ADAPTER IReactorData (* Adapter Interface *)
  (* Standard: 61499-1 *)
  (* Version 0.0, 7/4/2026, Schneider Electric *)
  PACKAGE SE.Nereda;
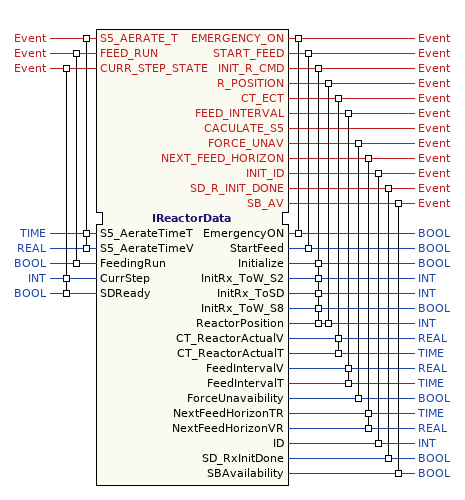
  EVENT_INPUT
    S5_AERATE_T WITH S5_AerateTimeT, S5_AerateTimeV;
    FEED_RUN WITH FeedingRun;
    CURR_STEP_STATE WITH CurrStep, SDReady;
  END_EVENT
  EVENT_OUTPUT
    EMERGENCY_ON WITH EmergencyON;
    START_FEED WITH StartFeed;
    INIT_R_CMD WITH ReactorPosition, Initialize, InitRx_ToW_S2, InitRx_ToSD, InitRx_ToW_S8;
    R_POSITION WITH ReactorPosition;
    CT_ECT WITH CT_ReactorActualV, CT_ReactorActualT;
    FEED_INTERVAL WITH FeedIntervalV, FeedIntervalT;
    CACULATE_S5;
    FORCE_UNAV WITH ForceUnavaibility;
    NEXT_FEED_HORIZON WITH NextFeedHorizonTR, NextFeedHorizonVR;
    INIT_ID WITH ID;
    SD_R_INIT_DONE WITH SD_RxInitDone;
    SB_AV WITH SBAvailability;
  END_EVENT
  VAR_INPUT
    S5_AerateTimeT : TIME;
    S5_AerateTimeV : REAL;
    FeedingRun : BOOL;
    CurrStep : INT;
    SDReady : BOOL;
  END_VAR
  VAR_OUTPUT
    EmergencyON : BOOL;
    StartFeed : BOOL;
    Initialize : BOOL;
    InitRx_ToW_S2 : INT;
    InitRx_ToSD : INT;
    InitRx_ToW_S8 : BOOL;
    ReactorPosition : INT;
    CT_ReactorActualV : REAL;
    CT_ReactorActualT : TIME;
    FeedIntervalV : REAL;
    FeedIntervalT : TIME;
    ForceUnavaibility : BOOL;
    NextFeedHorizonTR : TIME;
    NextFeedHorizonVR : REAL;
    ID : INT;
    SD_RxInitDone : BOOL;
    SBAvailability : BOOL;
  END_VAR
  SERVICE SOCKET/PLUG
    SEQUENCE request_confirm
      SOCKET.REQ(REQD) -> PLUG.REQ(REQD);
      PLUG.CNF(CNFD) -> SOCKET.CNF(CNFD);
    END_SEQUENCE
    SEQUENCE indication_response
      PLUG.IND(INDD) -> SOCKET.IND(INDD);
      SOCKET.RSP(RSPD) -> PLUG.RSP(RSPD);
    END_SEQUENCE
  END_SERVICE
END_ADAPTER
